// TIA Portal V17 export
// export: Created 2024-09-02T12:50:29.6384863Z, ExportSetting WithDefaults, DisplayName Totally Integrated Automation Portal, DisplayVersion V17, DisplayName TIA Portal Openness, DisplayVersion V17, DisplayName TIA Portal Version Control Interface, DisplayVersion V17, DisplayName STEP 7 Professional, DisplayVersion V17, DisplayName STEP 7 Safety, DisplayVersion V17, DisplayName WinCC Professional, DisplayVersion V17
TYPE "a_MGB"
// stored: IsFailsafeCompliant false
   STRUCT
      LedStart : Bool;   // Busmodul - LED Start / Bus module - LED start
      "res0.1" : Bool;   // Busmodul - Reserve / Bus module - reserve
      "res0.2" : Bool;   // Busmodul - Reserve / Bus module - reserve
      "res0.3" : Bool;   // Busmodul - Reserve / Bus module - reserve
      "res0.4" : Bool;   // Busmodul - Reserve / Bus module - reserve
      LedQuitt : Bool;   // Busmodul - LED Öffnen/Schliessen / Bus module - LED open/close
      "res0.6" : Bool;   // Busmodul - Reserve / Bus module - reserve
      "res0.7" : Bool;   // Busmodul - Reserve / Bus module - reserve
   END_STRUCT;
END_TYPE
